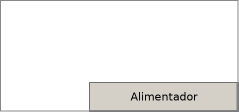
VISUALIZATION VS_FMS205_Test  // 239x112
VAR_IN_OUT
	
END_VAR
VAR
	TestAlimentador
END_VAR
    Button (89,82 150x30), "Alimentador"
        toggle MAIN.fbFMS205_Test.TestAlimentador
END_VISUALIZATION

(* stored: Version 1.1.0.1, ProductVersion 3.1.4024.11
   Visu VS_FMS205_Test: Id {53b82e9a-fb8a-4ef1-ba19-b0c14e561bee} *)
